RoboDK station: python_coding.rdk

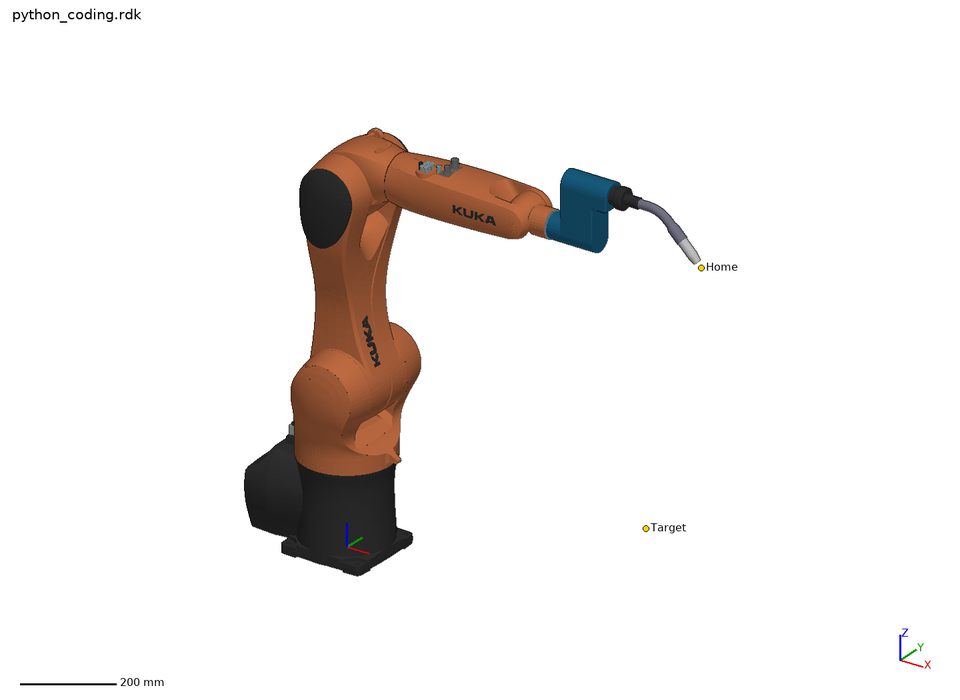
[picture v0: the station drawn from its stored meshes, robots at their saved joint values, targets as dots, program paths as lines]
Station python_coding (saved by RoboDK 5.6.8). Poses are relative to the parent item; angles as X-Y-Z fixed-axis rotations.
  - frame KUKA KR 6 R900 sixx Base at (0, 0, 0) mm
    - robot KUKA KR 6 R900 sixx: 6 axes, payload 6 kg, reach 901 mm, repeatability 0.03 mm, weight 52 kg
        modified DH rows (alpha deg, a mm, theta deg, d mm): 0, 0, 0, 400; -90, 25, 0, 0; 0, 455, -90, 0; -90, 35, 0, 420; 90, 0, 0, 0; -90, 0, 180, 80
        joint limits [-170, -190, -120, -185, -120, -350] to [170, 45, 156, 185, 120, 350]; home [0, -90, 90, 0, 0, 0]; saved at [0, -90, 90, 0, 0, 0]
      - tool Generic Welding Gun (Over-arm), TCP at (-4, 0, 371.3) mm, rotated rx 0 ry 45 rz 0 deg, size 169.7 x 60 x 367 mm
    - target Home (Cartesian target) at (896.3, 0, 894) mm, rotated rx -180 ry 45 rz -180 deg; joints [0, -90, 90, 0, 0, 0] of KUKA KR 6 R900 sixx
    - target Target (Cartesian target) at (756.3, 0, 254) mm, rotated rx 180 ry -15 rz -180 deg; joints [0, -73.67, 105.811, 0, 27.859, 0] of KUKA KR 6 R900 sixx
  - Python program Prog1 (listed below)

--- Python program Prog1 ---
# Type help("robodk.robolink") or help("robodk.robomath") for more information
# Press F5 to run the script
# Documentation: https://robodk.com/doc/en/RoboDK-API.html
# Reference:     https://robodk.com/doc/en/PythonAPI/robodk.html
# Note: It is not required to keep a copy of this file, your Python script is saved with your RDK project
#9le use of the RoboDK API:
# Remove these 2 lines to follow python programming guidelines
from robodk import *      # RoboDK API
from robolink import *    # Robot toolbox
# Link to RoboDK
RDK = Robolink()

# get the robot item:
robot = RDK.Item("KUKA KR 6 R900 sixx")

# get the home and target
home = RDK.Item("Home")
target = RDK.Item("Target")

# get the pose of the target (4x4 matrix)
poseref = target.Pose()
#print(poseref)


#move the robot to home, then to center :
robot.MoveJ(home)
robot.MoveJ(target)

# make an gexagon around the center:
for i in range(9):
    ang = i*2*pi/8
    posei = poseref*rotz(ang)*transl(100,0,0)*rotz(-ang)
    print(posei)
    robot.MoveL(posei)

# move back to the center, then home:
robot.MoveL(target)
robot.MoveJ(home)
